{attribute 'qualified_only'}
{attribute 'strict'}
TYPE E_EpicsHomeCmd :
    // Defines the valid options for homing in FB_MotionStage
(
    LOW_LIMIT := 1, // Low limit switch
    HIGH_LIMIT := 2, // High limit switch
    HOME_VIA_LOW := 3, // Home switch via low switch
    HOME_VIA_HIGH := 4, // Home switch via high switch
    ABSOLUTE_SET := 15, // Set here to be fHomePosition
    // MCS2
    AUTOZERO := -1,
    CURRENT_POSITION_METHOD := 37,
    NONE := -99 // Do not home, ever
) INT := NONE;
END_TYPE

(* stored: Version 1.1.0.1
   DUT E_EpicsHomeCmd: Id {97391387-6673-4061-a135-1a0002888344} *)
